(* Logix 5000 project; controller Add_On_Analog Emulate 5570 rev 33.11; software revision 33.00 *)

TASK MainTask (continuous, watchdog 500 ms) : MainProgram

MODULES
   Local : Emulate 5570 (ICP 2, rev 33.11)
      Sensors : vendor 1 type 12 code 20 (ICP 3, Ethernet SensorNet, rev 2.1)
         Process_Sensors : ETHERNET-MODULE (Ethernet Process, rev 1.1, Output RPI 10 ms)
END_MODULES

PROGRAM MainProgram   (* main routine MainRoutine *)

ROUTINE MainRoutine   (* ladder *)
   0: ;
END_ROUTINE
END_PROGRAM
